FUNCTION_BLOCK Konstanta_2 (* Composite FB wrapping other FBs *)
  (* Standard: 61499-2; Description: 2nd constant finder of ellipse fitting stiction-detection method *)
  (* Version 1.0, 2020-08-15, Candra Wardaya, UGM *)
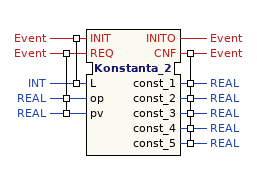
  EVENT_INPUT
    INIT WITH L; (* Initialization Request *)
    REQ WITH op, pv; (* Normal Execution Request *)
  END_EVENT
  EVENT_OUTPUT
    INITO; (* Initialization Confirm *)
    CNF WITH const_1, const_2, const_3, const_4, const_5; (* Execution Confirmation *)
  END_EVENT
  VAR_INPUT
    L : INT := 512; (* Array Length *)
    op : REAL; (* Controller Output Data *)
    pv : REAL; (* Process Variable Data *)
  END_VAR
  VAR_OUTPUT
    const_1 : REAL; (* Constant 1 *)
    const_2 : REAL; (* Constant 2 *)
    const_3 : REAL; (* Constant 3 *)
    const_4 : REAL; (* Constant 4 *)
    const_5 : REAL; (* Constant 5 *)
  END_VAR
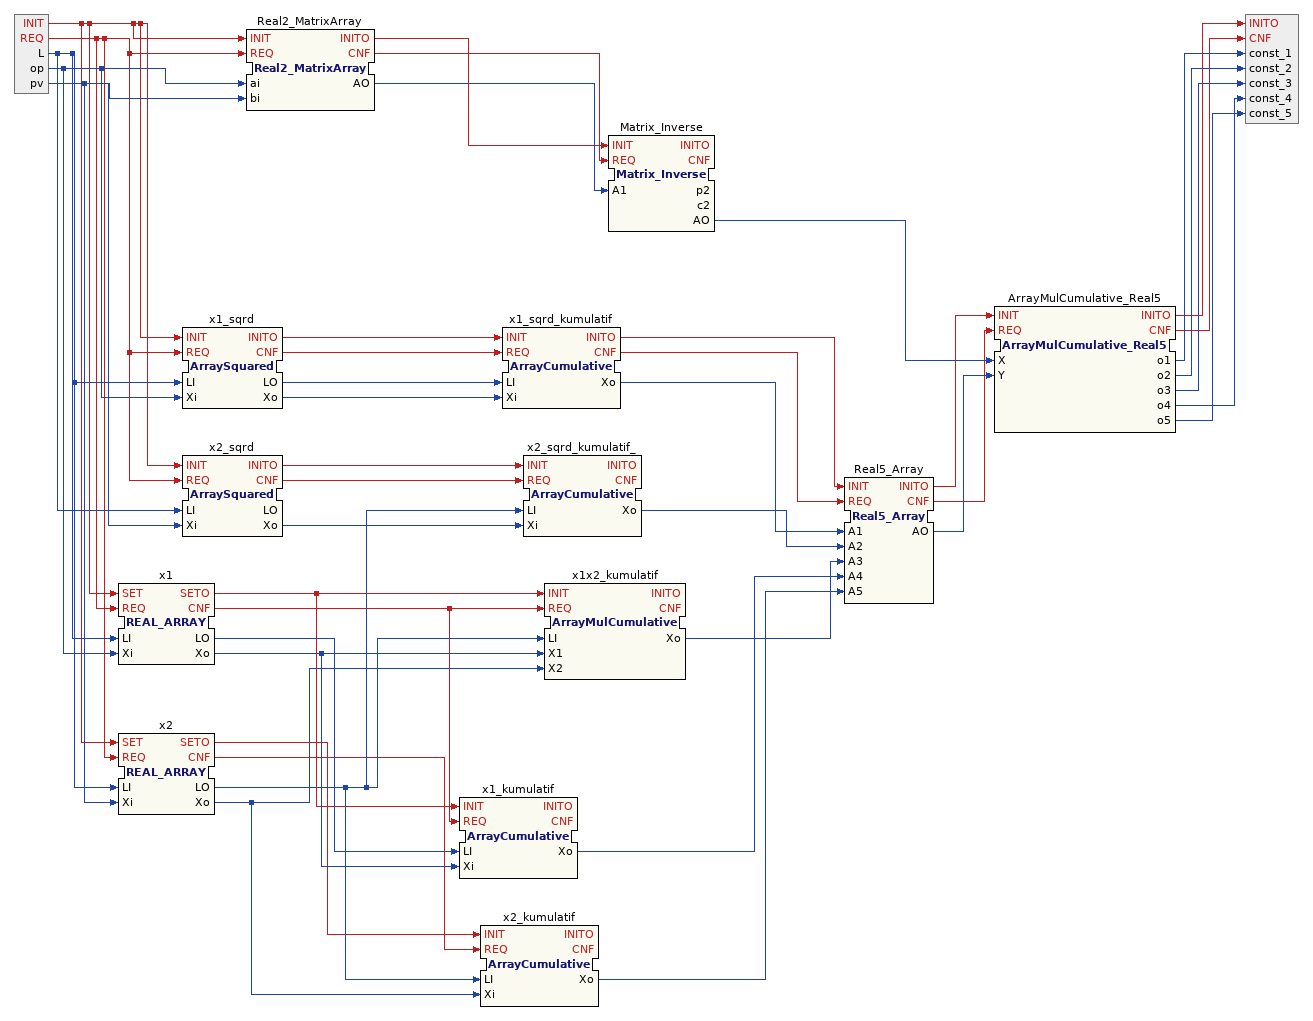
  FBS
    x2_sqrd_kumulatif_ : ArrayCumulative;
    x1_sqrd_kumulatif : ArrayCumulative;
    Real5_Array : Real5_Array;
    Real2_MatrixArray : Real2_MatrixArray;
    x1x2_kumulatif : ArrayMulCumulative;
    Matrix_Inverse : Matrix_Inverse;
    ArrayMulCumulative_Real5 : ArrayMulCumulative_Real5;
    x2_kumulatif : ArrayCumulative;
    x1_sqrd : ArraySquared;
    x2_sqrd : ArraySquared;
    x1_kumulatif : ArrayCumulative;
    x1 : REAL_ARRAY;
    x2 : REAL_ARRAY;
  END_FBS
  EVENT_CONNECTIONS
    x1_sqrd.CNF TO x1_sqrd_kumulatif.REQ;
    x1_sqrd_kumulatif.CNF TO Real5_Array.REQ;
    Real5_Array.INITO TO ArrayMulCumulative_Real5.INIT;
    Real2_MatrixArray.INITO TO Matrix_Inverse.INIT;
    x2_sqrd.CNF TO x2_sqrd_kumulatif_.REQ;
    x1_sqrd.INITO TO x1_sqrd_kumulatif.INIT;
    Real2_MatrixArray.CNF TO Matrix_Inverse.REQ;
    Real5_Array.CNF TO ArrayMulCumulative_Real5.REQ;
    x2_sqrd.INITO TO x2_sqrd_kumulatif_.INIT;
    x1_sqrd_kumulatif.INITO TO Real5_Array.INIT;
    INIT TO Real2_MatrixArray.INIT;
    INIT TO x1_sqrd.INIT;
    INIT TO x2_sqrd.INIT;
    REQ TO x1_sqrd.REQ;
    REQ TO x2_sqrd.REQ;
    REQ TO Real2_MatrixArray.REQ;
    ArrayMulCumulative_Real5.INITO TO INITO;
    ArrayMulCumulative_Real5.CNF TO CNF;
    INIT TO x1.SET;
    REQ TO x1.REQ;
    x1.SETO TO x1_kumulatif.INIT;
    x1.SETO TO x1x2_kumulatif.INIT;
    x1.CNF TO x1_kumulatif.REQ;
    x1.CNF TO x1x2_kumulatif.REQ;
    INIT TO x2.SET;
    REQ TO x2.REQ;
    x2.SETO TO x2_kumulatif.INIT;
    x2.CNF TO x2_kumulatif.REQ;
  END_CONNECTIONS
  DATA_CONNECTIONS
    x1_kumulatif.Xo TO Real5_Array.A4;
    x2_sqrd_kumulatif_.Xo TO Real5_Array.A2;
    Real5_Array.AO TO ArrayMulCumulative_Real5.Y;
    Matrix_Inverse.AO TO ArrayMulCumulative_Real5.X;
    x2_sqrd.Xo TO x2_sqrd_kumulatif_.Xi;
    Real2_MatrixArray.AO TO Matrix_Inverse.A1;
    x1x2_kumulatif.Xo TO Real5_Array.A3;
    x2_kumulatif.Xo TO Real5_Array.A5;
    x1_sqrd.Xo TO x1_sqrd_kumulatif.Xi;
    x1_sqrd_kumulatif.Xo TO Real5_Array.A1;
    op TO x1_sqrd.Xi;
    pv TO x2_sqrd.Xi;
    op TO Real2_MatrixArray.ai;
    pv TO Real2_MatrixArray.bi;
    ArrayMulCumulative_Real5.o1 TO const_1;
    ArrayMulCumulative_Real5.o2 TO const_2;
    ArrayMulCumulative_Real5.o3 TO const_3;
    ArrayMulCumulative_Real5.o4 TO const_4;
    ArrayMulCumulative_Real5.o5 TO const_5;
    L TO x1_sqrd.LI;
    L TO x2_sqrd.LI;
    x1_sqrd.LO TO x1_sqrd_kumulatif.LI;
    op TO x1.Xi;
    x1.Xo TO x1_kumulatif.Xi;
    x1.Xo TO x1x2_kumulatif.X1;
    pv TO x2.Xi;
    x2.Xo TO x2_kumulatif.Xi;
    x2.Xo TO x1x2_kumulatif.X2;
    L TO x1.LI;
    L TO x2.LI;
    x1.LO TO x1_kumulatif.LI;
    x2.LO TO x2_kumulatif.LI;
    x2.LO TO x1x2_kumulatif.LI;
    x2.LO TO x2_sqrd_kumulatif_.LI;
  END_CONNECTIONS
END_FUNCTION_BLOCK
